PROGRAM Auswertung_Alt
VAR
	platzhalter 		:BOOL;
	Switch				:BOOL;
END_VAR

// Auswertung der Leitung
	MAIN.Leitung.P_Leitung := MAIN.CW.Leitung;

// Auswertung ob Sekundär-Reaktor (Starten von GF_Befüllen)
IF Switch THEN
	ACT_GF_Befuellen();
	MAIN.Befuellen.M_START();
END_IF
// Prüfen ob GF_Entleeren
IF MAIN.CW.Enlteermenge > 0 THEN
	ACT_GF_Entleeren();
	MAIN.Entleeren.M_START();
END_IF
// Prüfen ob GF_Pumpen
IF MAIN.CW.Pumpmenge > 0 THEN
	ACT_GF_Pumpen();
	MAIN.Pumpen.M_START();
END_IF
// Prüfen ob GF_Halten
IF MAIN.CW.Haltedauer > T#0S THEN
	platzhalter := TRUE;
END_IF
// Prüfen ob GF_Rühren
IF MAIN.CW.Ruehrdauer > T#0S THEN
	ACT_GF_Ruehren();
	MAIN.Ruehren.M_START();
END_IF
// Prüfen ob GF_Warten
IF MAIN.CW.Wartedauer > T#0S THEN
	ACT_GF_Warten();
	MAIN.Warten.M_START();
END_IF
// Prüfen ob GF_Zirkulieren
IF MAIN.CW.Zirkulierdauer > T#0S THEN
	ACT_GF_Zirkulieren();
	MAIN.Zirkulieren.M_START();
END_IF

ACTION ACT_GF_Befuellen:
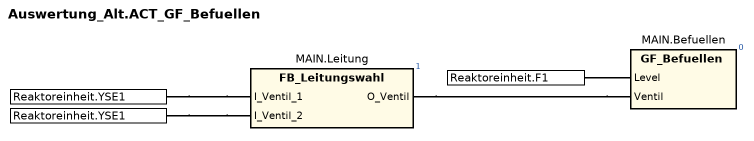
MAIN.Befuellen(Level := Reaktoreinheit.F1, Ventil := MAIN.Leitung.O_Ventil); // GF_Befuellen
MAIN.Leitung(I_Ventil_1 := Reaktoreinheit.YSE1, I_Ventil_2 := Reaktoreinheit.YSE1); // FB_Leitungswahl
END_ACTION

ACTION ACT_GF_Entleeren:
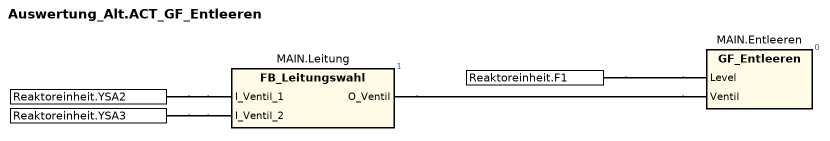
MAIN.Entleeren(Level := Reaktoreinheit.F1, Ventil := MAIN.Leitung.O_Ventil); // GF_Entleeren
MAIN.Leitung(I_Ventil_1 := Reaktoreinheit.YSA2, I_Ventil_2 := Reaktoreinheit.YSA3); // FB_Leitungswahl
END_ACTION

ACTION ACT_GF_Pumpen:
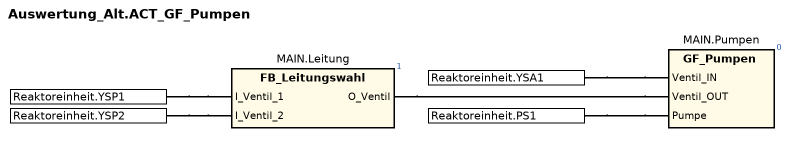
MAIN.Pumpen(
    Ventil_IN := Reaktoreinheit.YSA1,
    Ventil_OUT := MAIN.Leitung.O_Ventil,
    Pumpe := Reaktoreinheit.PS1); // GF_Pumpen
MAIN.Leitung(I_Ventil_1 := Reaktoreinheit.YSP1, I_Ventil_2 := Reaktoreinheit.YSP2); // FB_Leitungswahl
END_ACTION

ACTION ACT_GF_Ruehren:
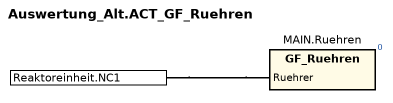
MAIN.Ruehren(Ruehrer := Reaktoreinheit.NC1); // GF_Ruehren
END_ACTION

ACTION ACT_GF_Warten:
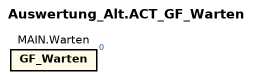
MAIN.Warten(); // GF_Warten
END_ACTION

ACTION ACT_GF_Zirkulieren:
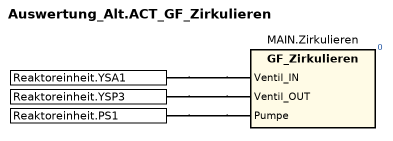
MAIN.Zirkulieren(
    Ventil_IN := Reaktoreinheit.YSA1,
    Ventil_OUT := Reaktoreinheit.YSP3,
    Pumpe := Reaktoreinheit.PS1); // GF_Zirkulieren
END_ACTION

END_PROGRAM

(* stored: Version 1.1.0.1, ProductVersion 3.1.4024.12
   POU Auswertung_Alt: Id {000f909d-068f-4416-91e8-93f170d3c0eb}, SpecialFunc None
   Action ACT_GF_Befuellen: Id {ae99807c-17fb-47fd-86b4-e2e6b43f0d43}
   Action ACT_GF_Entleeren: Id {f12b47ea-37bd-4410-b6f5-19e0ffdb3674}
   Action ACT_GF_Pumpen: Id {8f323d44-65ac-4ec7-b1ff-f8dab606d8f4}
   Action ACT_GF_Ruehren: Id {c551d848-7459-4181-8dee-6a9670d1da01}
   Action ACT_GF_Warten: Id {7d54961b-4edc-44c8-a047-8bcd95f023cb}
   Action ACT_GF_Zirkulieren: Id {a763afa8-a95e-4955-8282-6e3850ee7e64} *)
